TYPE DUT_LidChecking :
STRUCT
	arCameraResult:ARRAY[1..4,1..12] OF INT;
END_STRUCT
END_TYPE

(* stored: Version 1.1.0.1, ProductVersion 3.1.4024.9
   DUT DUT_LidChecking: Id {dd42250d-022e-45a6-ada8-fd56d1c9a980} *)
